// TwinCAT 3 PLC project PLC
// ProgramVersion: 3.1.4024.0
// libraries:
//   Tc2_Standard, * (Beckhoff Automation GmbH)
//   Tc2_System, * (Beckhoff Automation GmbH)
//   Tc3_BoolCounter, * (TE140x Module Vendor)
//   Tc3_Module, * (Beckhoff Automation GmbH)
// project tree:
//   / PlcTask.TcTTO
//   POUs/ MAIN.TcPOU
// real-time tasks:
//   TASK PlcTask: cycle T#10ms, priority 20, ADS port 350

CONFIGURATION PLC
    RESOURCE PLC ON TwinCAT3
        TASK PlcTask(INTERVAL := T#10ms, PRIORITY := 20);
        PROGRAM MAIN WITH PlcTask : MAIN;
    END_RESOURCE
END_CONFIGURATION

// ---- POUs/MAIN.TcPOU
PROGRAM MAIN
VAR CONSTANT
	Dimension1_Bools	: DINT	:= 3;
	Dimension2_Bools	: DINT	:= 4;
	Dimension1_Floats	: DINT	:= 6;
	Dimension2_Floats	: DINT	:= 2;
END_VAR
VAR
	fbCountBools			: FB_count_and_invert_booleans := ();
	Count					: LREAL;
	ArrayBools		AT %I*	: ARRAY[1..Dimension1_Bools, 1..Dimension2_Bools] OF BOOL	:= [7(TRUE)];
	InverseArray	AT %Q*	: ARRAY[1..Dimension1_Floats, 1..Dimension2_Floats] OF LREAL;
	o1						: DINT;
	o2						: DINT;
END_VAR

//Setting the input boolArray
fbCountBools.put_boolArray(data := ADR(ArrayBools), size1 := Dimension1_Bools, size2 := Dimension2_Bools);
//setting the input inverseArray
fbCountBools.put_inverseArray(data := ADR(InverseArray), size1 := Dimension1_Floats, size2 := Dimension2_Floats);
//execute the function
fbCountBools(fcount => Count);
o1	:= Dimension1_Floats;
o2	:= Dimension2_Floats;
//Getting the output inverseArray
fbCountBools.get_inverseArray_(data := ADR(InverseArray), size1 := o1, size2 := o2);

END_PROGRAM
